(*
SPDX-FileCopyrightText: © 2026 Oleksandr Tiutyk <trofimich@gmail.com>
SPDX-License-Identifier: MIT
License: https://opensource.org/license/mit
*)

(*!
<summary>Reports a field or property whose named type is not supported by the operation.</summary>
<description>
The caller detects the member error; Throw records diagnostics rather than inspecting the object. Dynamic
instances and clones belong to the current task memory manager until cleanup.
</description>
*)
INTERFACE IDataMemberTypeNotSupportedException EXTENDS IGeneralException

(*!
<summary>Formats the rejected member and propagates the exception.</summary>
<description>
Call in the owning cyclic task, not during FB_init. Builds a member diagnostic and captures source and
timestamps with zero error code and no inner cause. Input storage is not retained. Allocation failure uses the
shared terminal memory mechanism.
</description>
<param name="dataMemberName">Name of the field or property rejected by the caller.</param>
<param name="dataMemberTypeName">Name of the unsupported concrete type.</param>
*)
METHOD Throw
VAR_INPUT
	sourceNamespaceName : STRING;
	sourceClassName : STRING;
	sourcePOUName : STRING;
	sourcePosition : STRING;
	dataMemberName : STRING;
	dataMemberTypeName : STRING;
END_VAR
END_METHOD

END_INTERFACE

(* stored: Version 1.1.0.1
   Itf IDataMemberTypeNotSupportedException: Id {11c08bf0-c6ce-49fe-8b89-9f8f5e6c5095}
   Method Throw: Id {d75368a2-4715-4ba7-89d0-da1934b67c1e} *)
